// TIA Portal V19 export
FUNCTION_BLOCK "LKinAxisCtrl_Main"   // FB1, LAD
{ S7_Optimized_Access := 'TRUE' }
// stored: AutoNumber false, MemoryReserve 100, SetENOAutomatically false
   VAR_INPUT
      FirstCycle : Bool;
      StateSafetyActive : Bool := TRUE;
      StateInfeedInOperation : Bool;
      Power { ExternalAccessible := 'False'; ExternalVisible := 'False'; ExternalWritable := 'False'} : Bool;   // enable axis
      Reset { ExternalAccessible := 'False'; ExternalVisible := 'False'; ExternalWritable := 'False'} : Bool;   // reset axis
      Home { ExternalAccessible := 'False'; ExternalVisible := 'False'; ExternalWritable := 'False'} : Bool;   // Home axis / home axis
      Stop : Bool;
      Data : "LKinAxisCtrl_TypeDataParameters";
   END_VAR
   VAR_OUTPUT
      AxisPowered : Bool;
      AxisHomed : Bool;
      AxisError : Bool;
      ErrorProgram : Bool;
      KinematicError : Bool;
      KinematicInterrupted : Bool;
      AxisActualPosition : Array[1..6] of Real;
      KinematicActualPosition : Array[1..6] of Real;
      KinematicActualVelocity : Real;
      Diagnostics : Struct
         Status : Word;
         SubFunctionStatus : Word;
      END_STRUCT;
   END_VAR
   VAR_IN_OUT
      Robot : TO_Kinematics;
   END_VAR
   VAR
      statReadyForOperation : Bool;
      statFirstError : Bool;
      instLKinCtrl_MC_GroupPower { S7_SetPoint := 'True'} : "LKinCtrl_MC_GroupPower";
      instLKinCtrl_MC_GroupReset { S7_SetPoint := 'True'} : "LKinCtrl_MC_GroupReset";
      InstLKinCtrl_MC_GroupHome { S7_SetPoint := 'True'} : "LKinCtrl_MC_GroupHome";
      instLKinAxisCtrl_GroupPowered { S7_SetPoint := 'True'} : "LKinAxisCtrl_GroupPowered";
      instLKinAxisCtrl_GroupHomed { S7_SetPoint := 'True'} : "LKinAxisCtrl_GroupHomed";
      instLKinAxisCtrl_GroupError { S7_SetPoint := 'True'} : "LKinAxisCtrl_GroupError";
      "instLKinAxisCtrl_GroupPos&Velo" { S7_SetPoint := 'True'} : "LKinAxisCtrl_GroupPos&Velo";
      instLKinCtrl_GetKinematicsStatusWord { S7_SetPoint := 'True'} : "LKinCtrl_GetKinematicsStatusWord";
      instMC_GROUPSTOP { S7_SetPoint := 'True'} : MC_GROUPSTOP;
   END_VAR
   VAR_TEMP
      tempLreal : LReal;
   END_VAR
   VAR CONSTANT
      ERR_SAFETY : Word := 16#820C;
      ERR_INFEED : Word := 16#820D;
      ERR_COM_SENSOR : Word := 16#820E;
      ERR_COM_DRIVE : Word := 16#820F;
      ERR_MC_POWER : Word := 16#8600;
      ERR_MC_RESET : Word := 16#8601;
      ERR_MC_HOME : Word := 16#8602;
      ERR_MC_STOP : Word := 16#8603;
   END_VAR
BEGIN

REGION Network 1 (SCL): Test conditions for ready operation
   // Test conditions for ready operation
   //----------------------------------------------------------------------------------------------
   IF #StateSafetyActive AND #AxisPowered THEN
       #statFirstError := TRUE;
       #Diagnostics.Status := #ERR_SAFETY;
       #Diagnostics.SubFunctionStatus := 0;
   ELSIF NOT #StateInfeedInOperation AND #AxisPowered  THEN
       #statFirstError := TRUE;
       #Diagnostics.Status := #ERR_INFEED;
       #Diagnostics.SubFunctionStatus := 0;
   END_IF;
END_REGION

REGION Network 2: Drive Ready for Operation
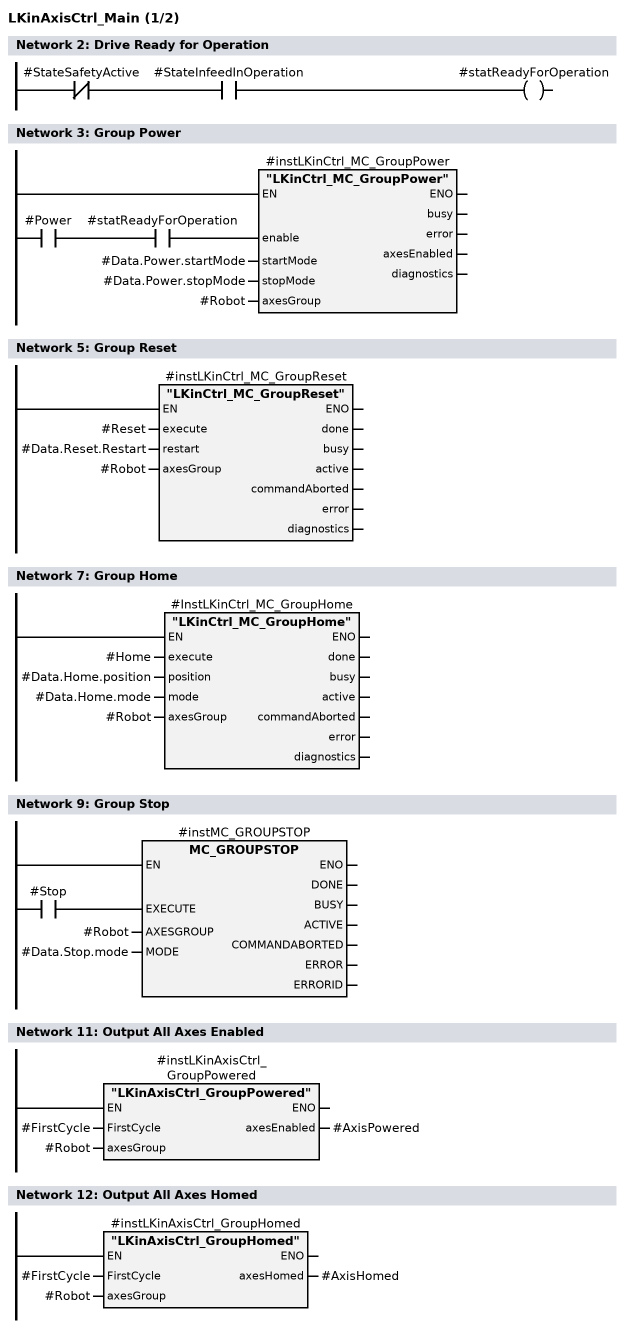
   RUNG wire#powerrail
      I_Contact( #StateSafetyActive )
      Contact( #StateInfeedInOperation )
      Coil( #statReadyForOperation )
   END_RUNG
   // the same network as SCL:
   #statReadyForOperation := NOT #StateSafetyActive AND #StateInfeedInOperation;
END_REGION

REGION Network 3: Group Power
   RUNG wire#powerrail
      #instLKinCtrl_MC_GroupPower(enable := wire#w1, startMode := #Data.Power.startMode, stopMode := #Data.Power.stopMode, axesGroup := #Robot, busy =>, error =>, axesEnabled =>, diagnostics =>)
   END_RUNG
   RUNG wire#powerrail
      Contact( #Power )
      Contact( #statReadyForOperation )
   END_RUNG wire#w1
   // the same network as SCL:
   #instLKinCtrl_MC_GroupPower(enable := #Power AND #statReadyForOperation,   // "LKinCtrl_MC_GroupPower"
                           startMode := #Data.Power.startMode,
                           stopMode := #Data.Power.stopMode,
                           axesGroup := #Robot);
END_REGION

REGION Network 4 (SCL): Test Return functions Power
   // MC_POWER
   IF (#instLKinCtrl_MC_GroupPower.error = TRUE) AND NOT #statFirstError THEN
       #statFirstError := TRUE;
       #Diagnostics.Status := #ERR_MC_POWER;
       #Diagnostics.SubFunctionStatus := #instLKinCtrl_MC_GroupPower.diagnostics.status;
   END_IF;
END_REGION

REGION Network 5: Group Reset
   RUNG wire#powerrail
      #instLKinCtrl_MC_GroupReset(execute := #Reset, restart := #Data.Reset.Restart, axesGroup := #Robot, done =>, busy =>, active =>, commandAborted =>, error =>, diagnostics =>)
   END_RUNG
   // the same network as SCL:
   #instLKinCtrl_MC_GroupReset(execute := #Reset, restart := #Data.Reset.Restart, axesGroup := #Robot);   // "LKinCtrl_MC_GroupReset"
END_REGION

REGION Network 6 (SCL): Test Return functions Reset
   // MC_RESET
   IF (#instLKinCtrl_MC_GroupReset.error = TRUE) AND NOT #statFirstError THEN
       #statFirstError := TRUE;
       #Diagnostics.Status := #ERR_MC_RESET;
       #Diagnostics.SubFunctionStatus := #instLKinCtrl_MC_GroupReset.diagnostics.status;
   END_IF;
END_REGION

REGION Network 7: Group Home
   RUNG wire#powerrail
      #InstLKinCtrl_MC_GroupHome(execute := #Home, position := #Data.Home.position, mode := #Data.Home.mode, axesGroup := #Robot, done =>, busy =>, active =>, commandAborted =>, error =>, diagnostics =>)
   END_RUNG
   // the same network as SCL:
   #InstLKinCtrl_MC_GroupHome(execute := #Home,   // "LKinCtrl_MC_GroupHome"
                           position := #Data.Home.position,
                           mode := #Data.Home.mode,
                           axesGroup := #Robot);
END_REGION

REGION Network 8 (SCL): Test Return functions Home
   // MC_HOME
   IF (#InstLKinCtrl_MC_GroupHome.error = TRUE) AND NOT #statFirstError THEN
       #statFirstError := TRUE;
       #Diagnostics.Status := #ERR_MC_HOME;
       #Diagnostics.SubFunctionStatus := #InstLKinCtrl_MC_GroupHome.diagnostics.status;
   END_IF;
END_REGION

REGION Network 9: Group Stop
   RUNG wire#powerrail
      #instMC_GROUPSTOP.MC_GROUPSTOP(Execute := wire#w1, AxesGroup := #Robot, Mode := #Data.Stop.mode, Done =>, Busy =>, Active =>, CommandAborted =>, Error =>, ErrorId =>)
   END_RUNG
   RUNG wire#powerrail
      Contact( #Stop )
   END_RUNG wire#w1
   // the same network as SCL:
   #instMC_GROUPSTOP(Execute := #Stop, AxesGroup := #Robot, Mode := #Data.Stop.mode);   // MC_GROUPSTOP
END_REGION

REGION Network 10 (SCL): Test Return functions Home / Test Return functions Stop
   // MC_HOME
   IF (#instMC_GROUPSTOP.Error = TRUE) AND NOT #statFirstError THEN
       #statFirstError := TRUE;
       #Diagnostics.Status := #ERR_MC_STOP;
       #Diagnostics.SubFunctionStatus := #instMC_GROUPSTOP.ErrorId;
   END_IF;
END_REGION

REGION Network 11: Output All Axes Enabled
   RUNG wire#powerrail
      #instLKinAxisCtrl_GroupPowered(FirstCycle := #FirstCycle, axesGroup := #Robot, axesEnabled => #AxisPowered)
   END_RUNG
   // the same network as SCL:
   #instLKinAxisCtrl_GroupPowered(FirstCycle := #FirstCycle, axesGroup := #Robot, axesEnabled => #AxisPowered);   // "LKinAxisCtrl_GroupPowered"
END_REGION

REGION Network 12: Output All Axes Homed
   RUNG wire#powerrail
      #instLKinAxisCtrl_GroupHomed(FirstCycle := #FirstCycle, axesGroup := #Robot, axesHomed => #AxisHomed)
   END_RUNG
   // the same network as SCL:
   #instLKinAxisCtrl_GroupHomed(FirstCycle := #FirstCycle, axesGroup := #Robot, axesHomed => #AxisHomed);   // "LKinAxisCtrl_GroupHomed"
END_REGION

REGION Network 13: Output All Axes in error
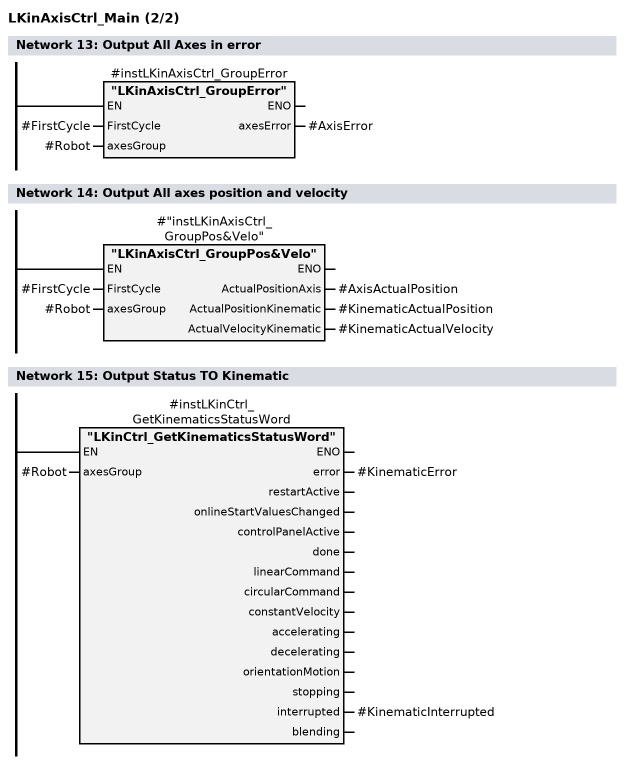
   RUNG wire#powerrail
      #instLKinAxisCtrl_GroupError(FirstCycle := #FirstCycle, axesGroup := #Robot, axesError => #AxisError)
   END_RUNG
   // the same network as SCL:
   #instLKinAxisCtrl_GroupError(FirstCycle := #FirstCycle, axesGroup := #Robot, axesError => #AxisError);   // "LKinAxisCtrl_GroupError"
END_REGION

REGION Network 14: Output All axes position and velocity
   RUNG wire#powerrail
      #"instLKinAxisCtrl_GroupPos&Velo"(FirstCycle := #FirstCycle, axesGroup := #Robot, ActualPositionAxis => #AxisActualPosition, ActualPositionKinematic => #KinematicActualPosition, ActualVelocityKinematic => #KinematicActualVelocity)
   END_RUNG
   // the same network as SCL:
   #"instLKinAxisCtrl_GroupPos&Velo"(FirstCycle := #FirstCycle,   // "LKinAxisCtrl_GroupPos&Velo"
                           axesGroup := #Robot,
                           ActualPositionAxis => #AxisActualPosition,
                           ActualPositionKinematic => #KinematicActualPosition,
                           ActualVelocityKinematic => #KinematicActualVelocity);
END_REGION

REGION Network 15: Output Status TO Kinematic
   RUNG wire#powerrail
      #instLKinCtrl_GetKinematicsStatusWord(axesGroup := #Robot, error => #KinematicError, restartActive =>, onlineStartValuesChanged =>, controlPanelActive =>, done =>, linearCommand =>, circularCommand =>, constantVelocity =>, accelerating =>, decelerating =>, orientationMotion =>, stopping =>, interrupted => #KinematicInterrupted, blending =>)
   END_RUNG
   // the same network as SCL:
   #instLKinCtrl_GetKinematicsStatusWord(axesGroup := #Robot,   // "LKinCtrl_GetKinematicsStatusWord"
                           error => #KinematicError,
                           interrupted => #KinematicInterrupted);
END_REGION

REGION Network 16 (SCL): Output Error state
   // Error state output
   //----------------------------------------------------------------------------------------------
   #ErrorProgram := #statFirstError;

   IF #Reset AND #statFirstError THEN
       #statFirstError := FALSE;
       #Diagnostics.Status := 0;
       #Diagnostics.SubFunctionStatus := 0;
   END_IF;
END_REGION
END_FUNCTION_BLOCK
